INTERFACE ITF_MCHMIPrepareScreen_00_05_Init

METHOD PUBLIC LinkDataHMI_00_05 : BOOL
VAR_INPUT
	refstData				: REFERENCE TO ST_MCHMIPrepareScreen_00_05;
END_VAR
END_METHOD

END_INTERFACE

(* stored: Version 1.1.0.1
   Itf ITF_MCHMIPrepareScreen_00_05_Init: Id {19f2fea5-18df-0cfe-2d12-9d47350bb28e}
   Method LinkDataHMI_00_05: Id {9b72961f-b481-0573-20bd-faffdd530a15} *)
